FUNCTION_BLOCK FB_VizuSIS
VAR_INPUT
	ATQ				: BOOL;
	RTQ				: BOOL;
	TTA				: BOOL;
	TDQ				: BOOL;
	TTA_Destination	: STRING(NAME_LENGTH) := '10-001-0100-01-1';
	PositionString	: STRING(NAME_LENGTH) := '10-001-0100-01-1'; // Name of position 11-111-1111-11-1;	
	ATQ_Dimension	: ST_Dimension :=(Width:=800, Length:=800, Height:=500, Weight:=1200);
	ATQ_Label		: STRING(Conveyor.LABEL_LENGTH) := 'CREATECODE';
	TU_ID			: STRING(Conveyor.TU_ID_STRINGLENGTH):= Conveyor.TU_ID_UNKNOWN; // TU-ID
	AssignmentID	: UDINT := Conveyor.ASSIGNMENT_ID_UNKNOWN;
	AutoID			: BOOL; //Use TU ID and Assignment ID from TU table for TTA and TDQ
END_VAR
VAR_OUTPUT
	BadPosition		: BOOL;
END_VAR
VAR
	myPos			: STRING(NAME_LENGTH);
	myTuIndex		: DINT;

	TrigATQ : R_TRIG();
	TrigRTQ : R_TRIG();
	TrigTTA : R_TRIG();
	TrigTDQ : R_TRIG();
	
END_VAR
VAR_TEMP
	Position : ST_PositionIdent;
END_VAR

myPos := F_ReduceToAlphaNumeric(PositionString);
Position := F_SearchFunctionPosition(Position := myPos);
BadPosition := Position.eFunctionNumber = E_FunctionNumber.F_BEGIN_FUNCTION;
IF(BadPosition) THEN
	RETURN;
END_IF


TrigATQ(CLK:=ATQ);
TrigRTQ(CLK:=RTQ);
TrigTTA(CLK:=TTA);
TrigTDQ(CLK:=TDQ);

IF(TrigATQ.Q) THEN
	//ATQDimension
	_M_SendATQ(Position,ATQ_Dimension,ATQ_Label);
	//F_AddPhysicalTU(Position.eFunctionNumber,Position.ZoneNumber);
END_IF

IF(TrigRTQ.Q) THEN
	F_RemovePhysicalTU(Position.eFunctionNumber,Position.ZoneNumber);
END_IF

IF(TrigTTA.Q) THEN	
	_M_SendTTA(Position,TTA_Destination,TU_ID,AssignmentID);
END_IF

IF(TrigTDQ.Q) THEN	
	_M_SendTDQ(Position);
END_IF

METHOD PRIVATE _M_GetIDs : BOOL
VAR_INPUT
	Position 		: REFERENCE TO ST_PositionIdent;	
	TU_ID			: REFERENCE TO STRING(Conveyor.TU_ID_STRINGLENGTH); // TU-ID
	AssigID			: REFERENCE TO UDINT ;
END_VAR

VAR
	myTuIndex		: DINT;
END_VAR
//(Conveyor.TU_ID_STRINGLENGTH):= Conveyor.TU_ID_UNKNOWN;
//:= Conveyor.ASSIGNMENT_ID_UNKNOWN

IF(THIS^.AutoID) THEN
	
	myTuIndex := F_PB_GetTransportControlDataRef(Position.eFunctionNumber,Position.ZoneNumber).TU_DataIndex;
	IF(myTuIndex>0) THEN
		AssigID		:= TU_Table.TU_DataTable[myTuIndex].AssignmentID;
		TU_ID 			:= TU_Table.TU_DataTable[myTuIndex].TU_ID.ASCII;
	ELSE
		AssigID 		:= Conveyor.ASSIGNMENT_ID_UNKNOWN;
		TU_ID		:= Conveyor.TU_ID_UNKNOWN;	
	END_IF	
ELSE
	//use the ID's from the input field of the vizio interface.
	TU_ID := THIS^.TU_ID;	
	AssigID := THIS^.AssignmentID;
END_IF
END_METHOD

METHOD PRIVATE _M_SendATQ : BOOL
VAR_INPUT
	Position 		: REFERENCE TO ST_PositionIdent;
	Dimension		: REFERENCE TO ST_Dimension;
	Label			: REFERENCE TO STRING(Conveyor.LABEL_LENGTH);	
END_VAR
VAR
	myLabel			: STRING(Conveyor.LABEL_LENGTH);
END_VAR
VAR_STAT
	ID		: INT := 1;
	ATQ		: ST_ITC_ATQ;
END_VAR

ATQ.Position := F_ReduceToAlphaNumeric(InputString := Position.PositionName);

IF(Label[0]=0) THEN

	myLabel := F_StuffString(
			InputString 	:= INT_TO_STRING(ID), 
			StringLength	:= 8, 
			StuffCharacter 	:= '0',
			LeftAligned     := FALSE);
	myLabel := CONCAT('TESTLABEL_',myLabel);
			
	ID := ID + 1;
	IF ID > 9998 THEN
		ID := 1;
	END_IF
ELSE
	myLabel := Label;
END_IF		

IF(Dimension.Height=0) THEN Dimension.Height:=200; END_IF
IF(Dimension.Length=0) THEN Dimension.Length:=200; END_IF
IF(Dimension.Weight=0) THEN Dimension.Weight:=200; END_IF
IF(Dimension.Width=0) THEN Dimension.Width:=200; END_IF

ATQ.Height := Dimension.Height;
ATQ.Length := Dimension.Length;
ATQ.Weight := Dimension.Weight;
ATQ.Width := Dimension.Width;

ATQ.LabelPresent := 1;
ATQ.Label := myLabel;


IF(ProBoxSystem.EMULATION_ENABLED) THEN
	fbITC_ManagerEmulation.M_AddData(
		meChannelSrc := 0,
		mMsgType     := E_ITC_MsgTypeConv.E_ADD_TU_REQUEST,
		mpData		 := ADR(ATQ),
		mLen 		 := SIZEOF(ATQ));
END_IF
END_METHOD

METHOD PRIVATE _M_SendTDQ : BOOL
VAR_INPUT
	Position 		: REFERENCE TO ST_PositionIdent;	
	//TU_Id    		: STRING(Conveyor.TU_ID_STRINGLENGTH);
END_VAR
VAR	
	TDQ		: ST_ITC_TDQ;
	
END_VAR

_M_GetIDs(Position,TDQ.TU_ID, TDQ.AssignmentID);

TDQ.Position := F_ReduceToAlphaNumeric(InputString := Position.PositionName);

TDQ.Code :=0;
TDQ.MsgSequence:=999;


_M_SendTDQ:= fbITC_Manager.M_AddData(
					meChannelSrc := 0,
					mMsgType     := E_ITC_MsgTypeConv.TASK_DELETE_REQUEST,
					mpData		 := ADR(TDQ),
					mLen		 := SIZEOF(TDQ));
END_METHOD

METHOD PRIVATE _M_SendTTA : BOOL
VAR_INPUT
	Position 		: REFERENCE TO ST_PositionIdent;
	Destination		: REFERENCE TO STRING(NAME_LENGTH);
	TU_Id    		: STRING(Conveyor.TU_ID_STRINGLENGTH);
	AssignmentID	: UDINT := Conveyor.ASSIGNMENT_ID_UNKNOWN;
END_VAR
VAR
	TTA		: ST_ITC_TTA;
	//mName	: STRING[NAME_LENGTH];
END_VAR
//mName := F_GetFunctionName(eFunctionNumber:= Position.eFunctionNumber, ZoneNumber:= Position.ZoneNumber);
TTA.Position := F_ReduceToAlphaNumeric(InputString := Position.PositionName);
//mName := F_GetFunctionName(eFunctionNumber:= Position.eFunctionNumber, ZoneNumber:= Position.ZoneNumber);
TTA.Destination[1] := F_ReduceToAlphaNumeric(InputString := Destination);//'11-001-0206-01-1';
TTA.DestinationSlot:=1;
TTA.NumberOfDestinations:=1;
TTA.AssignmentID:=AssignmentID;
TTA.TU_ID := TU_Id;

_M_GetIDs(Position,TTA.TU_ID, TTA.AssignmentID);

_M_SendTTA:= fbITC_Manager.M_AddData(
					meChannelSrc := 0,
					mMsgType     := E_ITC_MsgTypeConv.TRANSPORT_TASK_ASSIGNMENT,
					mpData		 := ADR(TTA),
					mLen		 := SIZEOF(TTA));
END_METHOD

END_FUNCTION_BLOCK

(* stored: Version 1.1.0.1, ProductVersion 3.1.4024.9
   POU FB_VizuSIS: Id {61ed0491-6ca7-4724-ab0b-28a94b94818a}, SpecialFunc None
   Method _M_GetIDs: Id {6e39bdf9-8700-4b47-8a91-d0c1a028c8ba}
   Method _M_SendATQ: Id {a4006221-e4c2-44d3-8c94-1c0c3d5307b4}
   Method _M_SendTDQ: Id {f44d007e-257e-42ff-99f6-1061e88daa4d}
   Method _M_SendTTA: Id {5ed76978-c2e8-4fd9-a492-01c533e6bd51} *)
